Yaskawa INFORM job: R1_W43-44-A2(80,180)KM-OK.JBI

/JOB
//NAME R1_W43-44-A2(80,180)KM-OK
///FOLDERNAME KRIS-SCIANA
//POS
///NPOS 89,89,0,2,0,0
///TOOL 0
///POSTYPE PULSE
///PULSE
C00000=13527,-43767,-75037,30600,77310,-61859
C00001=13527,-43767,-75037,30600,77310,-61859
C00002=110076,-43767,-75037,30600,77310,-61859
C00003=110076,-43767,-75037,30600,77310,-61859
C00004=123461,-43767,-75037,30600,77310,-61859
C00005=126362,-43170,-71794,29525,74883,-61447
C00006=127129,-43225,-69698,29356,73478,-61533
C00007=127483,-43162,-69660,29197,73370,-61428
C00008=126678,-42826,-70776,29441,74386,-61461
C00009=123408,-42240,-71618,30717,76222,-62146
C00010=128463,-10042,-58905,30625,91452,-59881
C00011=135733,-28551,-66517,20405,69729,-63965
C00012=135659,-28748,-64789,20593,68653,-64182
C00013=135585,-27921,-64222,20625,68744,-64193
C00014=135659,-28748,-64789,20593,68653,-64182
C00015=136878,-39110,-75133,19774,69363,-63638
C00016=133925,-57869,-75252,23872,58456,-58862
C00017=133925,-57972,-74870,23942,58193,-58923
C00018=133925,-57869,-75252,23872,58456,-58862
C00019=132786,-59261,-77041,24474,59128,-59170
C00020=129829,-62603,-81405,26003,60867,-59945
C00021=118853,-19899,-59266,40923,89558,-70743
C00022=121409,-21695,-57539,40075,86957,-70727
C00023=122378,-22670,-57593,39761,86187,-70633
C00024=122421,-21336,-57343,39736,86582,-70467
C00025=121353,-22353,-56800,40109,86365,-70974
C00026=122328,-16427,-52430,39777,86230,-70635
C00027=121387,-17374,-53940,40082,86970,-70732
C00028=118899,-15614,-55651,40907,89521,-70739
C00029=114095,-43801,-64911,56481,76171,59789
C00030=116620,-42818,-61164,56038,73692,59569
C00031=117498,-41786,-59660,55848,72960,59584
C00032=116643,-43720,-60589,56220,73209,59252
C00033=117612,-41689,-60442,55685,73203,59815
C00034=119264,-46764,-63016,55391,71659,59739
C00035=125682,-53702,-67426,50642,64091,62164
C00036=115467,-43883,-75441,54955,79154,62520
C00037=115467,-43883,-75441,54955,79154,62520
C00038=159887,-30519,-82518,-113,94753,49656
C00039=180385,-13971,-68139,-23942,109415,54550
C00040=179094,-19314,-68527,-23286,106803,54680
C00041=178707,-21879,-68930,-23047,105728,54773
C00042=179674,-21054,-68529,-23286,106119,55011
C00043=178424,-20149,-69044,-23130,106543,54515
C00044=179719,-19891,-67160,-23263,105904,55070
C00045=177430,-14751,-62619,-22768,105217,54460
C00046=180071,-17564,-66907,-23479,106946,54970
C00047=155437,-56075,-95332,-513,93890,31910
C00048=153193,-26490,-75152,3610,105634,32229
C00049=147441,-32400,-77587,10742,101859,31780
C00050=146986,-32855,-77735,10785,101632,31610
C00051=149258,-36624,-87368,10431,105310,32611
C00052=161583,-34538,-92851,-20048,109730,48661
C00053=143909,-124333,-126577,8064,53395,41899
C00054=26820,-112457,-122740,6292,56930,42963
C00055=62244,-61451,-105180,-7470,82879,44783
C00056=75644,-4460,-54939,-11618,88525,42492
C00057=56734,18444,-26661,8728,74038,25010
C00058=57572,19206,-23401,8362,72360,25160
C00059=58094,20890,-21375,8108,71932,25299
C00060=57489,19005,-23539,8407,72351,25132
C00061=58491,18035,-23493,7909,71737,25416
C00062=56829,16790,-22610,8831,70721,24802
C00063=56701,16618,-24264,8851,71654,24826
C00064=55847,15812,-27542,9218,73326,24674
C00065=51025,38559,-20408,11123,80987,-64845
C00066=58060,12439,-34607,-3071,60093,-66937
C00067=62074,19707,-20093,-6329,55124,-65280
C00068=62784,21670,-18237,-6882,55045,-65003
C00069=61644,18984,-23119,-5898,56577,-65522
C00070=57218,30457,-12012,-2584,55428,-67113
C00071=57609,32169,-8084,-2935,53905,-66927
C00072=58348,33826,-6375,-3519,53734,-66637
C00073=57238,25788,-19131,-2542,57410,-67156
C00074=54249,39015,-13309,12043,73677,-63833
C00075=58343,29181,-14560,4589,61267,-65070
C00076=54117,41744,-1786,7533,60158,-66625
C00077=46970,52437,-7513,15724,77991,-65580
C00078=46163,49298,-3084,16419,73954,-66369
C00079=47748,43981,64,15985,69179,-66501
C00080=50610,33288,-10917,14325,69905,-65430
C00081=50447,32650,-11282,14423,69838,-65494
C00082=50976,31235,-12304,14145,69659,-65337
C00083=48419,26796,-25664,15079,75823,-65409
C00084=55847,29330,-36998,8901,85942,25596
C00085=75566,-93497,-117956,-302,53023,30761
C00086=75566,-93497,-117956,1054,34216,30326
C00087=-3041,-146277,-132481,-3196,-9172,32117
C00088=-3041,-146277,-132481,-3196,-9172,32117
BC00000=255920,727322,1068222
BC00001=255920,727322,1068222
BC00002=393716,727322,1068222
BC00003=393716,1191142,1068222
BC00004=395053,1191142,1068222
BC00005=395053,1191142,1068222
BC00006=395053,1191142,1068222
BC00007=395053,1191142,1068222
BC00008=395053,1191142,1068222
BC00009=395053,1191142,1068222
BC00010=395053,1191142,1068222
BC00011=395053,1191142,1068222
BC00012=395053,1191142,1068222
BC00013=395053,1191142,1068222
BC00014=395053,1191142,1068222
BC00015=395053,1191142,1068222
BC00016=395053,1191142,1068222
BC00017=395053,1191142,1068222
BC00018=395053,1191142,1068222
BC00019=395053,1191142,1068222
BC00020=395053,1191142,1068222
BC00021=395053,1191142,1068222
BC00022=395053,1191142,1068222
BC00023=395053,1191142,1068222
BC00024=395053,1191142,1068222
BC00025=395053,1191142,1068222
BC00026=395053,1191142,1068222
BC00027=395053,1191142,1068222
BC00028=395053,1191142,1068222
BC00029=395053,1191142,1068222
BC00030=395053,1191142,1068222
BC00031=395053,1191142,1068222
BC00032=395053,1191142,1068222
BC00033=395053,1191142,1068222
BC00034=395053,1191142,1068222
BC00035=395053,1191142,1068222
BC00036=395053,1191142,1068222
BC00037=395053,1191142,1068222
BC00038=395053,1180258,1068222
BC00039=395053,1165292,1068222
BC00040=395053,1162385,1068222
BC00041=395053,1161221,1068216
BC00042=395053,1161222,1068222
BC00043=395053,1161222,1068222
BC00044=395053,1157770,1068222
BC00045=395053,1157770,1068222
BC00046=395053,1158932,1068222
BC00047=395053,1158932,1068222
BC00048=395053,1158932,1068222
BC00049=395053,1158932,1068222
BC00050=395053,1158932,1068222
BC00051=395053,1158932,1068222
BC00052=395053,1161839,1068222
BC00053=369197,1176903,1045669
BC00054=182681,1153482,1045669
BC00055=157788,1164947,1058085
BC00056=137464,1174307,1068222
BC00057=84161,1191142,1068222
BC00058=89742,1191142,1068222
BC00059=91969,1191142,1068222
BC00060=91975,1191142,1068222
BC00061=91975,1191142,1068222
BC00062=91942,1191142,1068222
BC00063=89709,1191142,1068222
BC00064=84128,1191142,1068222
BC00065=84128,1191142,1068222
BC00066=84128,1191142,1068222
BC00067=84128,1191142,1068222
BC00068=84128,1191142,1068222
BC00069=84128,1191142,1068222
BC00070=84128,1191142,1068222
BC00071=84128,1191142,1068222
BC00072=84128,1191142,1068222
BC00073=84128,1191142,1068222
BC00074=84128,1191142,1068222
BC00075=84128,1191142,1068222
BC00076=84128,1191142,1068222
BC00077=84128,1191142,1068222
BC00078=84128,1191142,1068222
BC00079=84128,1191142,1068222
BC00080=84128,1191142,1068222
BC00081=84128,1191142,1068221
BC00082=84128,1191142,1068221
BC00083=84128,1191142,1068221
BC00084=84128,1191142,1068222
BC00085=84128,1191142,1068222
BC00086=84128,1191142,1068222
BC00087=21207,1191142,1068222
BC00088=21207,693392,1068222
///POSTYPE BASE
///RECTAN
///RCONF 0,0,0,0,0,0,0,0,0,0,0,0,0,0,0,0,0,0,0,0,0,0,0,0
P00006=0.222,-3.123,-1.508,0.0000,0.0000,0.0000
P00023=0.143,-0.036,0.682,0.0000,0.0000,0.0000
//INST
///DATE 2024/07/25 11:53
///ATTR SC,RW
///GROUP1 RB1,BS1
NOP
'r1_W43-44-A2(80,180)
'Path S1263
SFTOF
MOVJ C00000 BC00000 VJ=100.00
MOVJ C00001 BC00001 VJ=100.00
MOVJ C00002 BC00002 VJ=100.00
MOVJ C00003 BC00003 VJ=100.00
MOVJ C00004 BC00004 VJ=100.00
MOVJ C00005 BC00005 VJ=20.00
MOVL C00006 BC00006 V=60.0
REFP 3 C00007 BC00007
CALL JOB:SEARCH-R1
SET P023 P006
SFTON P023
MOVL C00008 BC00008 V=60.0
MOVJ C00009 BC00009 VJ=20.00
MOVL C00010 BC00010 V=60.0
MOVL C00011 BC00011 V=83.3
MOVL C00012 BC00012 V=83.3
REFP 3 C00013 BC00013
CALL JOB:SEARCH-R1
SET P023 P006
SFTON P023
MOVL C00014 BC00014 V=83.3
MOVL C00015 BC00015 V=83.3
MOVL C00016 BC00016 V=60.0
REFP 3 C00017 BC00017
CALL JOB:SEARCH-R1
SET P023 P006
SFTON P023
MOVL C00018 BC00018 V=60.0
MOVL C00019 BC00019 V=166.7
MOVL C00020 BC00020 V=400.0
'Path W1265
SFTOF
SFTON P023
MOVJ C00021 BC00021 VJ=20.00
MOVJ C00022 BC00022 VJ=20.00
MOVL C00023 BC00023 V=100.0 PL=0
REFP 1 C00024 BC00024
REFP 2 C00025 BC00025
MACRO1 MJ#(0) ARGF7
ARCON
MOVL C00026 BC00026 V=10.8
ARCOF
MOVL C00027 BC00027 V=100.0
MOVL C00028 BC00028 V=166.7
SFTOF
'Path W1266
SFTOF
SFTON P023
MOVJ C00029 BC00029 VJ=20.00
MOVJ C00030 BC00030 VJ=20.00
MOVL C00031 BC00031 V=100.0 PL=0
REFP 1 C00032 BC00032
REFP 2 C00033 BC00033
MACRO1 MJ#(0) ARGF7
ARCON
MOVL C00034 BC00034 V=10.8
MOVL C00035 BC00035 V=10.8
ARCOF
MOVL C00036 BC00036 V=100.0
MOVL C00037 BC00037 V=166.7
SFTOF
'Path W1268
SFTOF
MOVJ C00038 BC00038 VJ=20.00
'Path W1269
SFTOF
SFTON P023
MOVJ C00039 BC00039 VJ=20.00
MOVJ C00040 BC00040 VJ=20.00
MOVL C00041 BC00041 V=100.0 PL=0
REFP 1 C00042 BC00042
REFP 2 C00043 BC00043
MACRO1 MJ#(0) ARGF7
ARCON
MOVL C00044 BC00044 V=10.8
MOVL C00045 BC00045 V=10.8
ARCOF
MOVL C00046 BC00046 V=100.0
MOVL C00047 BC00047 V=166.7
MOVL C00048 BC00048 V=166.7
ARCON
MOVL C00049 BC00049 V=10.0
MOVL C00050 BC00050 V=10.0
ARCOF
MOVL C00051 BC00051 V=166.7
SFTOF
'Path VIA1273
SFTOF
MOVJ C00052 BC00052 VJ=20.00
'Path VIA1274
SFTOF
MOVJ C00053 BC00053 VJ=20.00
'Path VIA1275
SFTOF
MOVJ C00054 BC00054 VJ=20.00
'Path W1270
SFTOF
SFTON P023
MOVJ C00055 BC00055 VJ=20.00
MOVJ C00056 BC00056 VJ=20.00
'Path W1271
SFTOF
SFTON P023
MOVJ C00057 BC00057 VJ=20.00
MOVJ C00058 BC00058 VJ=20.00
MOVL C00059 BC00059 V=100.0 PL=0
REFP 1 C00060 BC00060
REFP 2 C00061 BC00061
MACRO1 MJ#(0) ARGF7
ARCON
MOVL C00062 BC00062 V=10.0
ARCOF
MOVL C00063 BC00063 V=100.0
MOVL C00064 BC00064 V=166.7
MOVJ C00065 BC00065 VJ=20.00
MOVJ C00066 BC00066 VJ=10.00
MACRO1 MJ#(0) ARGF7
MOVJ C00067 BC00067 VJ=10.00
'ARCON
MOVL C00068 BC00068 V=10.8
'ARCOFF
MOVJ C00069 BC00069 VJ=10.00
MOVJ C00070 BC00070 VJ=10.00
MACRO1 MJ#(0) ARGF6
MOVJ C00071 BC00071 VJ=10.00
'ARCON
MOVL C00072 BC00072 V=10.0
'ARCOFF
MOVJ C00073 BC00073 VJ=10.00
SFTOF
MOVJ C00074 BC00074 VJ=20.00
SFTON P023
MACRO1 MJ#(0) ARGF7
MOVJ C00075 BC00075 VJ=20.00
ARCON
MOVL C00076 BC00076 V=7.5
ARCOF
MOVJ C00077 BC00077 VJ=20.00
MOVJ C00078 BC00078 VJ=10.00
MACRO1 MJ#(0) ARGF6
MOVJ C00079 BC00079 VJ=10.00
ARCON
TIMER T=0.20
ARCOF
MOVJ C00080 BC00080 VJ=10.00
ARCON
TIMER T=0.20
ARCOF
MOVJ C00081 BC00081 VJ=10.00
ARCON
MOVL C00082 BC00082 V=6.7
ARCOF
MOVJ C00083 BC00083 VJ=10.00
MOVJ C00084 BC00084 VJ=20.00
MOVJ C00085 BC00085 VJ=50.00
SFTOF
MOVJ C00086 BC00086 VJ=100.00
MOVJ C00087 BC00087 VJ=100.00
MOVJ C00088 BC00088 VJ=100.00
END
